// TIA Portal V17 export
// export: Created 2022-04-06T07:28:37.8382062Z, ExportSetting WithDefaults, DisplayName Totally Integrated Automation Portal, DisplayVersion V17, DisplayName TIA Portal Openness, DisplayVersion V17, DisplayName TIA Portal Version Control Interface, DisplayVersion V17, DisplayName TIA Portal Test Suite Advanced, DisplayVersion V17, DisplayName SINAMICS Startdrive Advanced, DisplayVersion V17, DisplayName SINAMICS Startdrive G130, G150, S120, S150, SINAMICS MV, S210, DisplayVersion V17, DisplayName SINAMICS Startdrive G110M, G120, G120C, G120D, G120P, G115D, DisplayVersion V17, DisplayName STEP 7 Professional, DisplayVersion V17, DisplayName STEP 7 Safety, DisplayVersion V17, DisplayName WinCC Advanced / Unified PC, DisplayVersion V17
FUNCTION_BLOCK "Main_Safety_RTG1"   // FB1, F_FBD
{ S7_Optimized_Access := 'TRUE' }
VERSION : 0.1
// stored: AutoNumber false, IsIECCheckEnabled false, UDAEnableTagReadback false
   VAR
      instACK_GL : ACK_GL;
      instLDrvSafe_SinaTlg901Control_1 : "LDrvSafe_typeSinaTlg901Control";
      instLDrvSafe_SinaTlg901Control : "LDrvSafe_SinaTlg901Control";
      instLDrvSafe_SinaTlg901Status : "LDrvSafe_SinaTlg901Status";
      instLDrvSafe_SinaSTlg30Control2 : "LDrvSafe_SinaSTlg30Control";
      instLDrvSafe_SinaSTlg30Status2 : "LDrvSafe_SinaSTlg30Status";
      instSINA_FFB : "SINA_FFB";
      instSINA_FFB1 : "SINA_FFB1";
   END_VAR
BEGIN

REGION Network 1
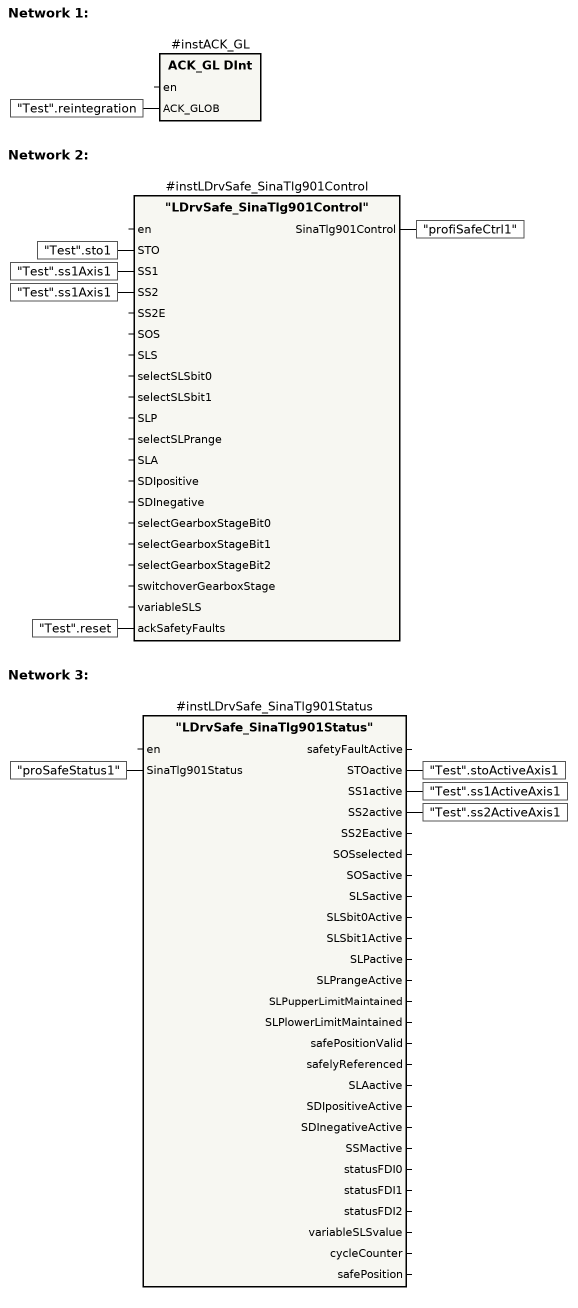
   #instACK_GL(ACK_GLOB := "Test".reintegration);   // ACK_GL
END_REGION

REGION Network 2
   #instLDrvSafe_SinaTlg901Control(STO := "Test".sto1,   // "LDrvSafe_SinaTlg901Control"
                           SS1 := "Test".ss1Axis1,
                           SS2 := "Test".ss1Axis1,
                           ackSafetyFaults := "Test".reset,
                           SinaTlg901Control => "profiSafeCtrl1");
END_REGION

REGION Network 3
   #instLDrvSafe_SinaTlg901Status(SinaTlg901Status := "proSafeStatus1",   // "LDrvSafe_SinaTlg901Status"
                           STOactive => "Test".stoActiveAxis1,
                           SS1active => "Test".ss1ActiveAxis1,
                           SS2active => "Test".ss2ActiveAxis1);
END_REGION

REGION Network 5
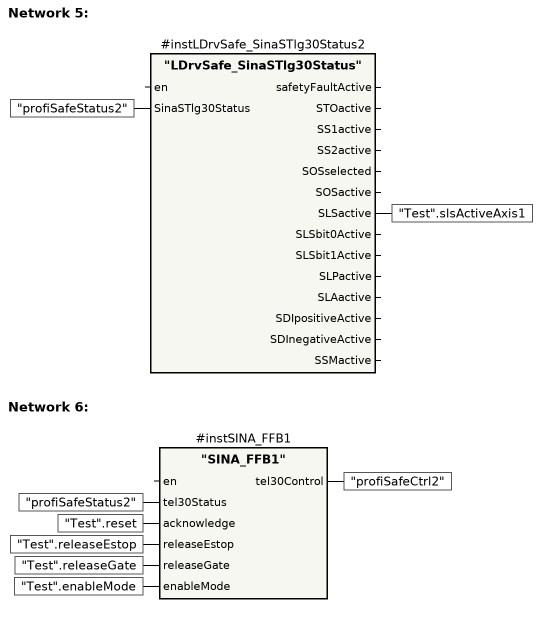
   #instLDrvSafe_SinaSTlg30Status2(SinaSTlg30Status := "profiSafeStatus2", SLSactive => "Test".slsActiveAxis1);   // "LDrvSafe_SinaSTlg30Status"
END_REGION

REGION Network 6
   #instSINA_FFB1(tel30Status := "profiSafeStatus2",   // "SINA_FFB1"
                  acknowledge := "Test".reset,
                  releaseEstop := "Test".releaseEstop,
                  releaseGate := "Test".releaseGate,
                  enableMode := "Test".enableMode,
                  tel30Control => "profiSafeCtrl2");
END_REGION
END_FUNCTION_BLOCK
